TEXTLIST TextList_Util_Defaut
  1 = 'Défaut' | FR: 'Droits par défaut' | EN: 'Rights by default'
   = ''
END_TEXTLIST

(* stored: Version 1.1.0.1, ProductVersion 3.1.4024.10
   TextList TextList_Util_Defaut: Id {18fd187e-898d-4d59-80f5-db789e34cecd} *)
